// TIA Portal V19 export
FUNCTION "Decoiler1_CALL" : Void   // FC129, LAD
TITLE = DECOILER 1 CALL
// stored: SetENOAutomatically false
   VAR_TEMP
      Feed_PB_InLine : "Ax_PB";
      Feed_PB_OutLine : "Ax_PB";
      Jaws_PB_InLine : "ValveMachine_PB";
      Jaws_PB_OutLine : "ValveMachine_PB";
      Coupling_PB_InLine : "ValveMachine_PB";
      Coupling_PB_OutLine : "ValveMachine_PB";
      SnubberLift_PB_InLine : "ValveMachine_PB";
      SnubberLift_PB_OutLine : "ValveMachine_PB";
      SnubberRoll_PB_InLine : "ValveMachine_PB";
      SnubberRoll_PB_OutLine : "ValveMachine_PB";
   END_VAR
BEGIN

REGION Network 1: Data In - PB Feed
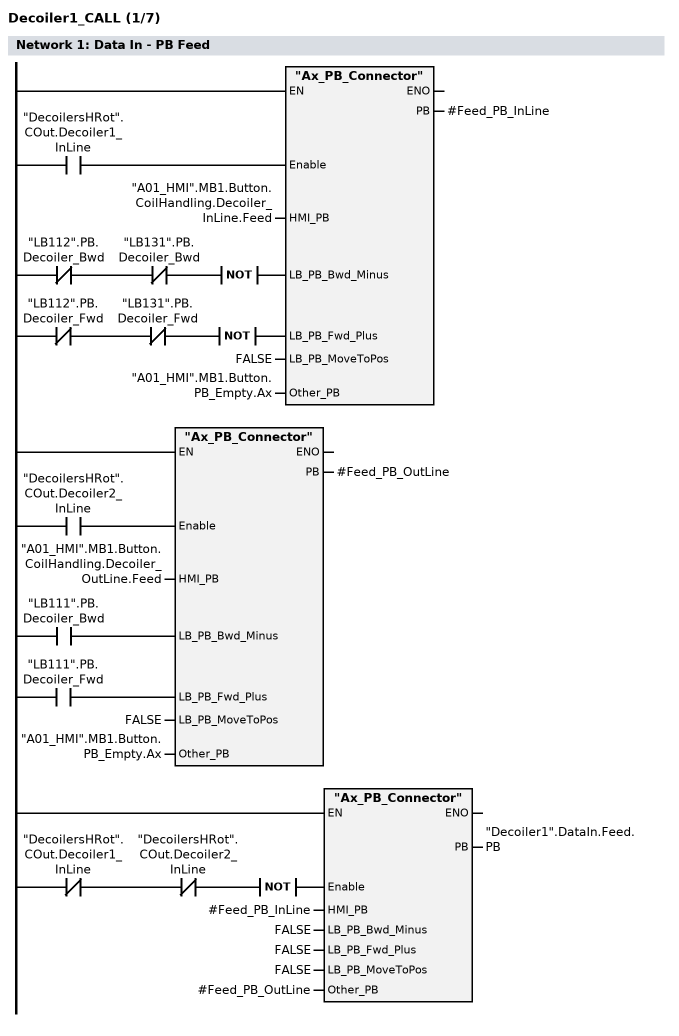
   RUNG wire#powerrail
      "Ax_PB_Connector"(Enable := wire#w1, LB_PB_Bwd_Minus := wire#w2, LB_PB_Fwd_Plus := wire#w3, HMI_PB := "A01_HMI".MB1.Button.CoilHandling.Decoiler_InLine.Feed, LB_PB_MoveToPos := FALSE, Other_PB := "A01_HMI".MB1.Button.PB_Empty.Ax, PB => #Feed_PB_InLine)
   END_RUNG
   RUNG wire#powerrail
      Contact( "DecoilersHRot".COut.Decoiler1_InLine )
   END_RUNG wire#w1
   RUNG wire#powerrail
      I_Contact( "LB112".PB.Decoiler_Bwd )
      I_Contact( "LB131".PB.Decoiler_Bwd )
      Not()
   END_RUNG wire#w2
   RUNG wire#powerrail
      I_Contact( "LB112".PB.Decoiler_Fwd )
      I_Contact( "LB131".PB.Decoiler_Fwd )
      Not()
   END_RUNG wire#w3
   RUNG wire#powerrail
      "Ax_PB_Connector"(Enable := wire#w4, LB_PB_Bwd_Minus := wire#w5, LB_PB_Fwd_Plus := wire#w6, HMI_PB := "A01_HMI".MB1.Button.CoilHandling.Decoiler_OutLine.Feed, LB_PB_MoveToPos := FALSE, Other_PB := "A01_HMI".MB1.Button.PB_Empty.Ax, PB => #Feed_PB_OutLine)
   END_RUNG
   RUNG wire#powerrail
      Contact( "DecoilersHRot".COut.Decoiler2_InLine )
   END_RUNG wire#w4
   RUNG wire#powerrail
      Contact( "LB111".PB.Decoiler_Bwd )
   END_RUNG wire#w5
   RUNG wire#powerrail
      Contact( "LB111".PB.Decoiler_Fwd )
   END_RUNG wire#w6
   RUNG wire#powerrail
      "Ax_PB_Connector"(Enable := wire#w7, HMI_PB := #Feed_PB_InLine, LB_PB_Bwd_Minus := FALSE, LB_PB_Fwd_Plus := FALSE, LB_PB_MoveToPos := FALSE, Other_PB := #Feed_PB_OutLine, PB => "Decoiler1".DataIn.Feed.PB)
   END_RUNG
   RUNG wire#powerrail
      I_Contact( "DecoilersHRot".COut.Decoiler1_InLine )
      I_Contact( "DecoilersHRot".COut.Decoiler2_InLine )
      Not()
   END_RUNG wire#w7
   // the same network as SCL:
   "Ax_PB_Connector"(Enable := "DecoilersHRot".COut.Decoiler1_InLine,
                     HMI_PB := "A01_HMI".MB1.Button.CoilHandling.Decoiler_InLine.Feed,
                     LB_PB_Bwd_Minus := NOT (NOT "LB112".PB.Decoiler_Bwd AND NOT "LB131".PB.Decoiler_Bwd),
                     LB_PB_Fwd_Plus := NOT (NOT "LB112".PB.Decoiler_Fwd AND NOT "LB131".PB.Decoiler_Fwd),
                     LB_PB_MoveToPos := FALSE,
                     Other_PB := "A01_HMI".MB1.Button.PB_Empty.Ax,
                     PB => #Feed_PB_InLine);
   "Ax_PB_Connector"(Enable := "DecoilersHRot".COut.Decoiler2_InLine,
                     HMI_PB := "A01_HMI".MB1.Button.CoilHandling.Decoiler_OutLine.Feed,
                     LB_PB_Bwd_Minus := "LB111".PB.Decoiler_Bwd,
                     LB_PB_Fwd_Plus := "LB111".PB.Decoiler_Fwd,
                     LB_PB_MoveToPos := FALSE,
                     Other_PB := "A01_HMI".MB1.Button.PB_Empty.Ax,
                     PB => #Feed_PB_OutLine);
   "Ax_PB_Connector"(Enable := NOT (NOT "DecoilersHRot".COut.Decoiler1_InLine AND NOT "DecoilersHRot".COut.Decoiler2_InLine),
                     HMI_PB := #Feed_PB_InLine,
                     LB_PB_Bwd_Minus := FALSE,
                     LB_PB_Fwd_Plus := FALSE,
                     LB_PB_MoveToPos := FALSE,
                     Other_PB := #Feed_PB_OutLine,
                     PB => "Decoiler1".DataIn.Feed.PB);
END_REGION

REGION Network 2: Data In - PB Jaws
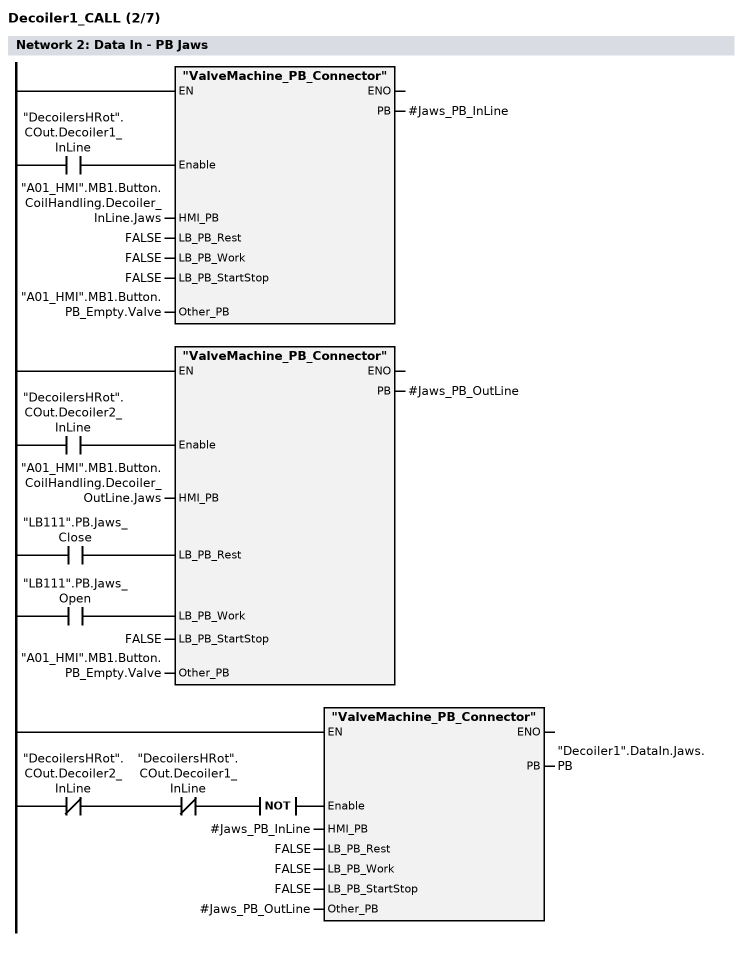
   RUNG wire#powerrail
      "ValveMachine_PB_Connector"(Enable := wire#w1, HMI_PB := "A01_HMI".MB1.Button.CoilHandling.Decoiler_InLine.Jaws, LB_PB_Rest := FALSE, LB_PB_Work := FALSE, LB_PB_StartStop := FALSE, Other_PB := "A01_HMI".MB1.Button.PB_Empty.Valve, PB => #Jaws_PB_InLine)
   END_RUNG
   RUNG wire#powerrail
      Contact( "DecoilersHRot".COut.Decoiler1_InLine )
   END_RUNG wire#w1
   RUNG wire#powerrail
      "ValveMachine_PB_Connector"(Enable := wire#w2, LB_PB_Rest := wire#w3, LB_PB_Work := wire#w4, HMI_PB := "A01_HMI".MB1.Button.CoilHandling.Decoiler_OutLine.Jaws, LB_PB_StartStop := FALSE, Other_PB := "A01_HMI".MB1.Button.PB_Empty.Valve, PB => #Jaws_PB_OutLine)
   END_RUNG
   RUNG wire#powerrail
      Contact( "DecoilersHRot".COut.Decoiler2_InLine )
   END_RUNG wire#w2
   RUNG wire#powerrail
      Contact( "LB111".PB.Jaws_Close )
   END_RUNG wire#w3
   RUNG wire#powerrail
      Contact( "LB111".PB.Jaws_Open )
   END_RUNG wire#w4
   RUNG wire#powerrail
      "ValveMachine_PB_Connector"(Enable := wire#w5, HMI_PB := #Jaws_PB_InLine, LB_PB_Rest := FALSE, LB_PB_Work := FALSE, LB_PB_StartStop := FALSE, Other_PB := #Jaws_PB_OutLine, PB => "Decoiler1".DataIn.Jaws.PB)
   END_RUNG
   RUNG wire#powerrail
      I_Contact( "DecoilersHRot".COut.Decoiler2_InLine )
      I_Contact( "DecoilersHRot".COut.Decoiler1_InLine )
      Not()
   END_RUNG wire#w5
   // the same network as SCL:
   "ValveMachine_PB_Connector"(Enable := "DecoilersHRot".COut.Decoiler1_InLine,
                           HMI_PB := "A01_HMI".MB1.Button.CoilHandling.Decoiler_InLine.Jaws,
                           LB_PB_Rest := FALSE,
                           LB_PB_Work := FALSE,
                           LB_PB_StartStop := FALSE,
                           Other_PB := "A01_HMI".MB1.Button.PB_Empty.Valve,
                           PB => #Jaws_PB_InLine);
   "ValveMachine_PB_Connector"(Enable := "DecoilersHRot".COut.Decoiler2_InLine,
                           HMI_PB := "A01_HMI".MB1.Button.CoilHandling.Decoiler_OutLine.Jaws,
                           LB_PB_Rest := "LB111".PB.Jaws_Close,
                           LB_PB_Work := "LB111".PB.Jaws_Open,
                           LB_PB_StartStop := FALSE,
                           Other_PB := "A01_HMI".MB1.Button.PB_Empty.Valve,
                           PB => #Jaws_PB_OutLine);
   "ValveMachine_PB_Connector"(Enable := NOT (NOT "DecoilersHRot".COut.Decoiler2_InLine AND NOT "DecoilersHRot".COut.Decoiler1_InLine),
                           HMI_PB := #Jaws_PB_InLine,
                           LB_PB_Rest := FALSE,
                           LB_PB_Work := FALSE,
                           LB_PB_StartStop := FALSE,
                           Other_PB := #Jaws_PB_OutLine,
                           PB => "Decoiler1".DataIn.Jaws.PB);
END_REGION

REGION Network 3: Data In - PB Couplung
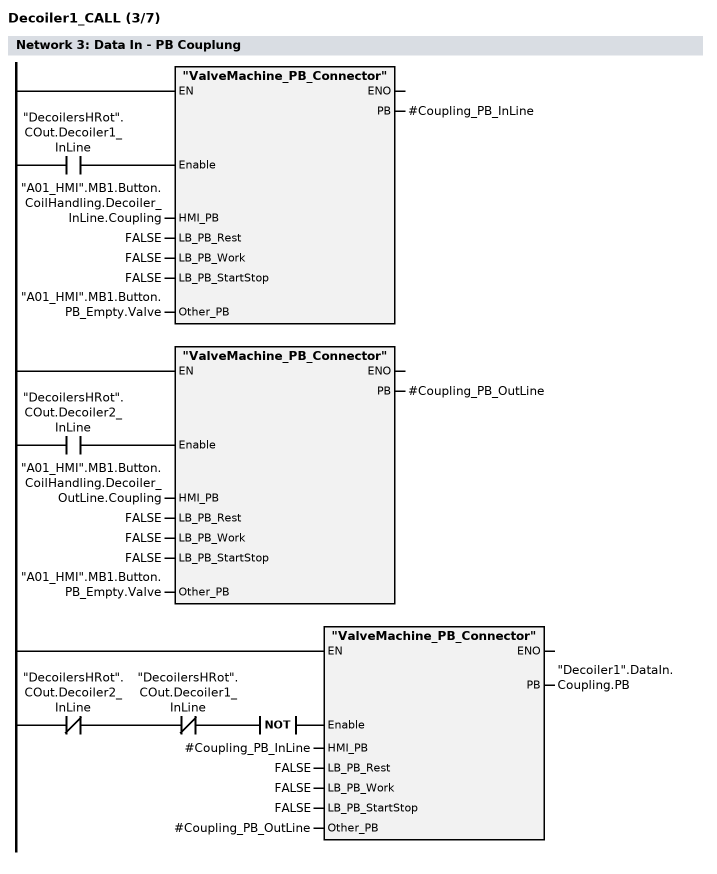
   RUNG wire#powerrail
      "ValveMachine_PB_Connector"(Enable := wire#w1, HMI_PB := "A01_HMI".MB1.Button.CoilHandling.Decoiler_InLine.Coupling, LB_PB_Rest := FALSE, LB_PB_Work := FALSE, LB_PB_StartStop := FALSE, Other_PB := "A01_HMI".MB1.Button.PB_Empty.Valve, PB => #Coupling_PB_InLine)
   END_RUNG
   RUNG wire#powerrail
      Contact( "DecoilersHRot".COut.Decoiler1_InLine )
   END_RUNG wire#w1
   RUNG wire#powerrail
      "ValveMachine_PB_Connector"(Enable := wire#w2, HMI_PB := "A01_HMI".MB1.Button.CoilHandling.Decoiler_OutLine.Coupling, LB_PB_Rest := FALSE, LB_PB_Work := FALSE, LB_PB_StartStop := FALSE, Other_PB := "A01_HMI".MB1.Button.PB_Empty.Valve, PB => #Coupling_PB_OutLine)
   END_RUNG
   RUNG wire#powerrail
      Contact( "DecoilersHRot".COut.Decoiler2_InLine )
   END_RUNG wire#w2
   RUNG wire#powerrail
      "ValveMachine_PB_Connector"(Enable := wire#w3, HMI_PB := #Coupling_PB_InLine, LB_PB_Rest := FALSE, LB_PB_Work := FALSE, LB_PB_StartStop := FALSE, Other_PB := #Coupling_PB_OutLine, PB => "Decoiler1".DataIn.Coupling.PB)
   END_RUNG
   RUNG wire#powerrail
      I_Contact( "DecoilersHRot".COut.Decoiler2_InLine )
      I_Contact( "DecoilersHRot".COut.Decoiler1_InLine )
      Not()
   END_RUNG wire#w3
   // the same network as SCL:
   "ValveMachine_PB_Connector"(Enable := "DecoilersHRot".COut.Decoiler1_InLine,
                           HMI_PB := "A01_HMI".MB1.Button.CoilHandling.Decoiler_InLine.Coupling,
                           LB_PB_Rest := FALSE,
                           LB_PB_Work := FALSE,
                           LB_PB_StartStop := FALSE,
                           Other_PB := "A01_HMI".MB1.Button.PB_Empty.Valve,
                           PB => #Coupling_PB_InLine);
   "ValveMachine_PB_Connector"(Enable := "DecoilersHRot".COut.Decoiler2_InLine,
                           HMI_PB := "A01_HMI".MB1.Button.CoilHandling.Decoiler_OutLine.Coupling,
                           LB_PB_Rest := FALSE,
                           LB_PB_Work := FALSE,
                           LB_PB_StartStop := FALSE,
                           Other_PB := "A01_HMI".MB1.Button.PB_Empty.Valve,
                           PB => #Coupling_PB_OutLine);
   "ValveMachine_PB_Connector"(Enable := NOT (NOT "DecoilersHRot".COut.Decoiler2_InLine AND NOT "DecoilersHRot".COut.Decoiler1_InLine),
                           HMI_PB := #Coupling_PB_InLine,
                           LB_PB_Rest := FALSE,
                           LB_PB_Work := FALSE,
                           LB_PB_StartStop := FALSE,
                           Other_PB := #Coupling_PB_OutLine,
                           PB => "Decoiler1".DataIn.Coupling.PB);
END_REGION

REGION Network 4: Data In - PB Snubber Lift
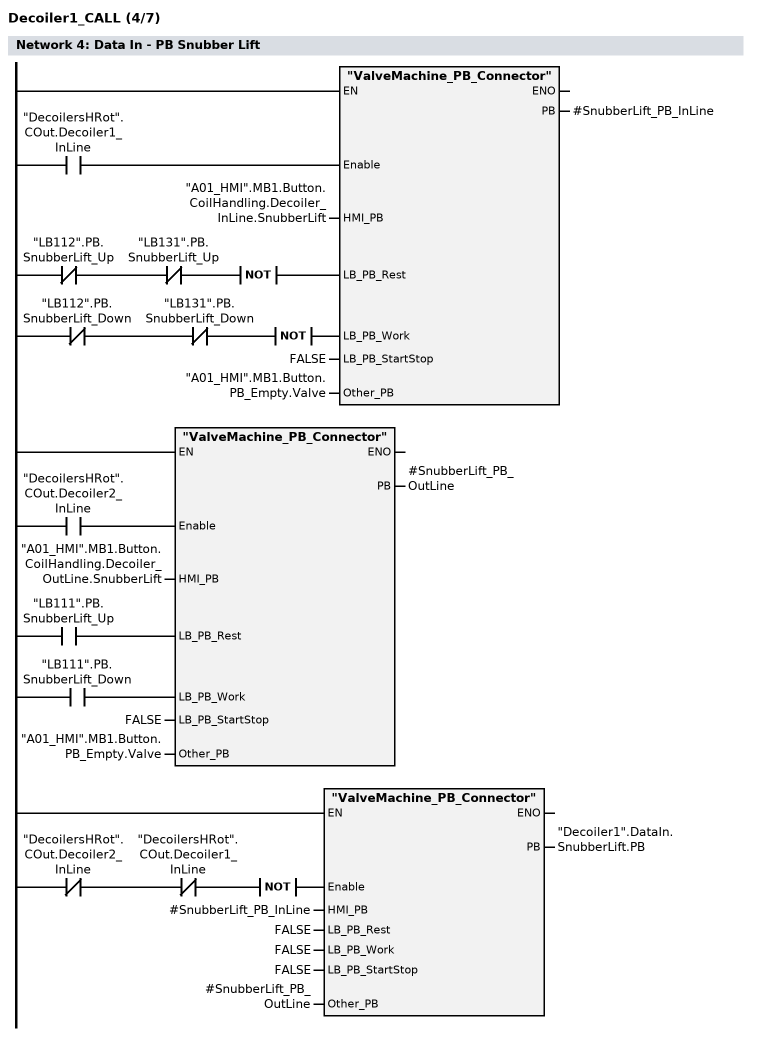
   RUNG wire#powerrail
      "ValveMachine_PB_Connector"(Enable := wire#w1, LB_PB_Rest := wire#w2, LB_PB_Work := wire#w3, HMI_PB := "A01_HMI".MB1.Button.CoilHandling.Decoiler_InLine.SnubberLift, LB_PB_StartStop := FALSE, Other_PB := "A01_HMI".MB1.Button.PB_Empty.Valve, PB => #SnubberLift_PB_InLine)
   END_RUNG
   RUNG wire#powerrail
      Contact( "DecoilersHRot".COut.Decoiler1_InLine )
   END_RUNG wire#w1
   RUNG wire#powerrail
      I_Contact( "LB112".PB.SnubberLift_Up )
      I_Contact( "LB131".PB.SnubberLift_Up )
      Not()
   END_RUNG wire#w2
   RUNG wire#powerrail
      I_Contact( "LB112".PB.SnubberLift_Down )
      I_Contact( "LB131".PB.SnubberLift_Down )
      Not()
   END_RUNG wire#w3
   RUNG wire#powerrail
      "ValveMachine_PB_Connector"(Enable := wire#w4, LB_PB_Rest := wire#w5, LB_PB_Work := wire#w6, HMI_PB := "A01_HMI".MB1.Button.CoilHandling.Decoiler_OutLine.SnubberLift, LB_PB_StartStop := FALSE, Other_PB := "A01_HMI".MB1.Button.PB_Empty.Valve, PB => #SnubberLift_PB_OutLine)
   END_RUNG
   RUNG wire#powerrail
      Contact( "DecoilersHRot".COut.Decoiler2_InLine )
   END_RUNG wire#w4
   RUNG wire#powerrail
      Contact( "LB111".PB.SnubberLift_Up )
   END_RUNG wire#w5
   RUNG wire#powerrail
      Contact( "LB111".PB.SnubberLift_Down )
   END_RUNG wire#w6
   RUNG wire#powerrail
      "ValveMachine_PB_Connector"(Enable := wire#w7, HMI_PB := #SnubberLift_PB_InLine, LB_PB_Rest := FALSE, LB_PB_Work := FALSE, LB_PB_StartStop := FALSE, Other_PB := #SnubberLift_PB_OutLine, PB => "Decoiler1".DataIn.SnubberLift.PB)
   END_RUNG
   RUNG wire#powerrail
      I_Contact( "DecoilersHRot".COut.Decoiler2_InLine )
      I_Contact( "DecoilersHRot".COut.Decoiler1_InLine )
      Not()
   END_RUNG wire#w7
   // the same network as SCL:
   "ValveMachine_PB_Connector"(Enable := "DecoilersHRot".COut.Decoiler1_InLine,
                           HMI_PB := "A01_HMI".MB1.Button.CoilHandling.Decoiler_InLine.SnubberLift,
                           LB_PB_Rest := NOT (NOT "LB112".PB.SnubberLift_Up AND NOT "LB131".PB.SnubberLift_Up),
                           LB_PB_Work := NOT (NOT "LB112".PB.SnubberLift_Down AND NOT "LB131".PB.SnubberLift_Down),
                           LB_PB_StartStop := FALSE,
                           Other_PB := "A01_HMI".MB1.Button.PB_Empty.Valve,
                           PB => #SnubberLift_PB_InLine);
   "ValveMachine_PB_Connector"(Enable := "DecoilersHRot".COut.Decoiler2_InLine,
                           HMI_PB := "A01_HMI".MB1.Button.CoilHandling.Decoiler_OutLine.SnubberLift,
                           LB_PB_Rest := "LB111".PB.SnubberLift_Up,
                           LB_PB_Work := "LB111".PB.SnubberLift_Down,
                           LB_PB_StartStop := FALSE,
                           Other_PB := "A01_HMI".MB1.Button.PB_Empty.Valve,
                           PB => #SnubberLift_PB_OutLine);
   "ValveMachine_PB_Connector"(Enable := NOT (NOT "DecoilersHRot".COut.Decoiler2_InLine AND NOT "DecoilersHRot".COut.Decoiler1_InLine),
                           HMI_PB := #SnubberLift_PB_InLine,
                           LB_PB_Rest := FALSE,
                           LB_PB_Work := FALSE,
                           LB_PB_StartStop := FALSE,
                           Other_PB := #SnubberLift_PB_OutLine,
                           PB => "Decoiler1".DataIn.SnubberLift.PB);
END_REGION

REGION Network 5: Data In - Snubber Roll
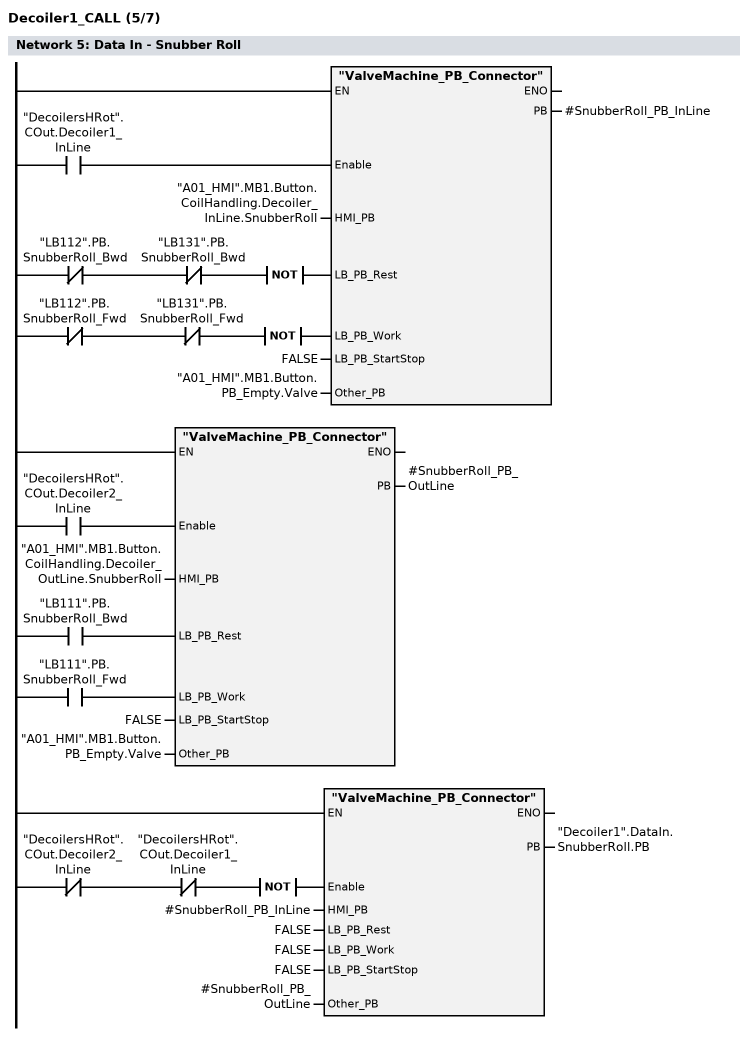
   RUNG wire#powerrail
      "ValveMachine_PB_Connector"(Enable := wire#w1, LB_PB_Rest := wire#w2, LB_PB_Work := wire#w3, HMI_PB := "A01_HMI".MB1.Button.CoilHandling.Decoiler_InLine.SnubberRoll, LB_PB_StartStop := FALSE, Other_PB := "A01_HMI".MB1.Button.PB_Empty.Valve, PB => #SnubberRoll_PB_InLine)
   END_RUNG
   RUNG wire#powerrail
      Contact( "DecoilersHRot".COut.Decoiler1_InLine )
   END_RUNG wire#w1
   RUNG wire#powerrail
      I_Contact( "LB112".PB.SnubberRoll_Bwd )
      I_Contact( "LB131".PB.SnubberRoll_Bwd )
      Not()
   END_RUNG wire#w2
   RUNG wire#powerrail
      I_Contact( "LB112".PB.SnubberRoll_Fwd )
      I_Contact( "LB131".PB.SnubberRoll_Fwd )
      Not()
   END_RUNG wire#w3
   RUNG wire#powerrail
      "ValveMachine_PB_Connector"(Enable := wire#w4, LB_PB_Rest := wire#w5, LB_PB_Work := wire#w6, HMI_PB := "A01_HMI".MB1.Button.CoilHandling.Decoiler_OutLine.SnubberRoll, LB_PB_StartStop := FALSE, Other_PB := "A01_HMI".MB1.Button.PB_Empty.Valve, PB => #SnubberRoll_PB_OutLine)
   END_RUNG
   RUNG wire#powerrail
      Contact( "DecoilersHRot".COut.Decoiler2_InLine )
   END_RUNG wire#w4
   RUNG wire#powerrail
      Contact( "LB111".PB.SnubberRoll_Bwd )
   END_RUNG wire#w5
   RUNG wire#powerrail
      Contact( "LB111".PB.SnubberRoll_Fwd )
   END_RUNG wire#w6
   RUNG wire#powerrail
      "ValveMachine_PB_Connector"(Enable := wire#w7, HMI_PB := #SnubberRoll_PB_InLine, LB_PB_Rest := FALSE, LB_PB_Work := FALSE, LB_PB_StartStop := FALSE, Other_PB := #SnubberRoll_PB_OutLine, PB => "Decoiler1".DataIn.SnubberRoll.PB)
   END_RUNG
   RUNG wire#powerrail
      I_Contact( "DecoilersHRot".COut.Decoiler2_InLine )
      I_Contact( "DecoilersHRot".COut.Decoiler1_InLine )
      Not()
   END_RUNG wire#w7
   // the same network as SCL:
   "ValveMachine_PB_Connector"(Enable := "DecoilersHRot".COut.Decoiler1_InLine,
                           HMI_PB := "A01_HMI".MB1.Button.CoilHandling.Decoiler_InLine.SnubberRoll,
                           LB_PB_Rest := NOT (NOT "LB112".PB.SnubberRoll_Bwd AND NOT "LB131".PB.SnubberRoll_Bwd),
                           LB_PB_Work := NOT (NOT "LB112".PB.SnubberRoll_Fwd AND NOT "LB131".PB.SnubberRoll_Fwd),
                           LB_PB_StartStop := FALSE,
                           Other_PB := "A01_HMI".MB1.Button.PB_Empty.Valve,
                           PB => #SnubberRoll_PB_InLine);
   "ValveMachine_PB_Connector"(Enable := "DecoilersHRot".COut.Decoiler2_InLine,
                           HMI_PB := "A01_HMI".MB1.Button.CoilHandling.Decoiler_OutLine.SnubberRoll,
                           LB_PB_Rest := "LB111".PB.SnubberRoll_Bwd,
                           LB_PB_Work := "LB111".PB.SnubberRoll_Fwd,
                           LB_PB_StartStop := FALSE,
                           Other_PB := "A01_HMI".MB1.Button.PB_Empty.Valve,
                           PB => #SnubberRoll_PB_OutLine);
   "ValveMachine_PB_Connector"(Enable := NOT (NOT "DecoilersHRot".COut.Decoiler2_InLine AND NOT "DecoilersHRot".COut.Decoiler1_InLine),
                           HMI_PB := #SnubberRoll_PB_InLine,
                           LB_PB_Rest := FALSE,
                           LB_PB_Work := FALSE,
                           LB_PB_StartStop := FALSE,
                           Other_PB := #SnubberRoll_PB_OutLine,
                           PB => "Decoiler1".DataIn.SnubberRoll.PB);
END_REGION

REGION Network 6: Data In - Pneumatic Brake
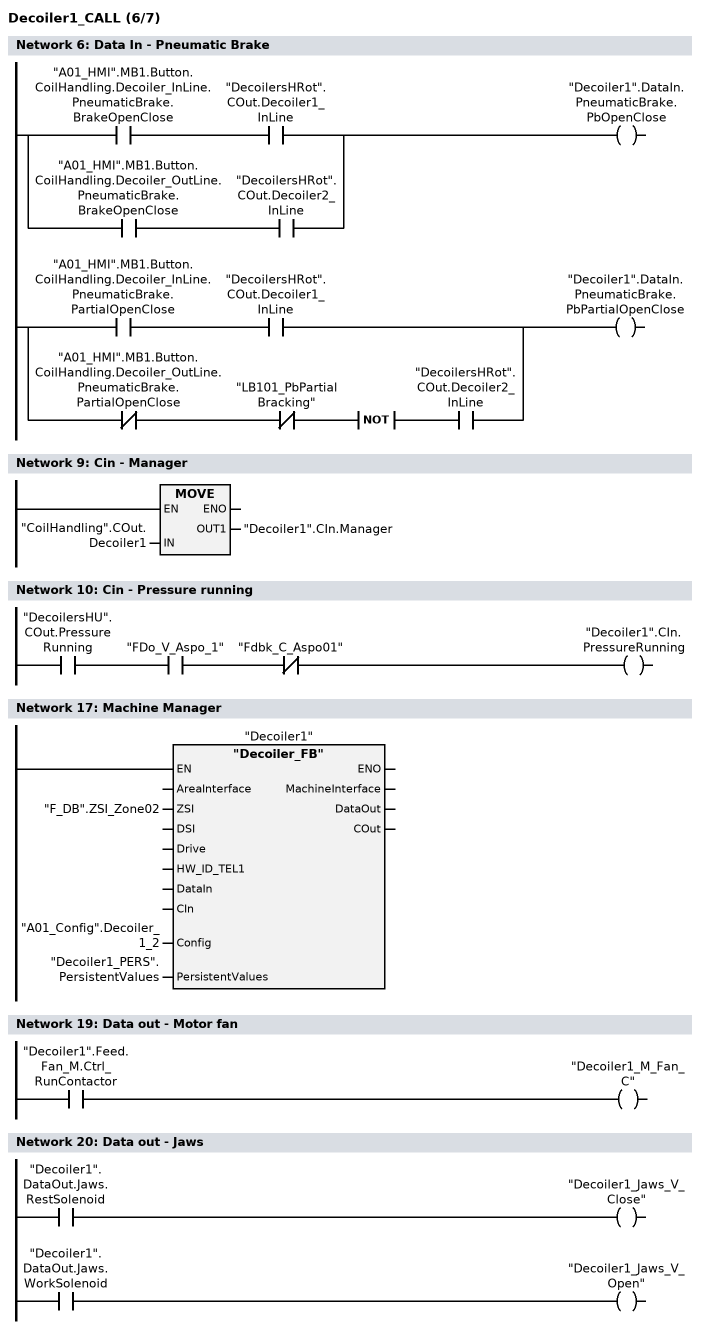
   RUNG wire#powerrail
      Contact( "A01_HMI".MB1.Button.CoilHandling.Decoiler_InLine.PneumaticBrake.BrakeOpenClose )
      Contact( "DecoilersHRot".COut.Decoiler1_InLine )
      wire#w1
      Coil( "Decoiler1".DataIn.PneumaticBrake.PbOpenClose )
   END_RUNG
   RUNG wire#powerrail
      Contact( "A01_HMI".MB1.Button.CoilHandling.Decoiler_OutLine.PneumaticBrake.BrakeOpenClose )
      Contact( "DecoilersHRot".COut.Decoiler2_InLine )
   END_RUNG wire#w1
   RUNG wire#powerrail
      Contact( "A01_HMI".MB1.Button.CoilHandling.Decoiler_InLine.PneumaticBrake.PartialOpenClose )
      Contact( "DecoilersHRot".COut.Decoiler1_InLine )
      wire#w2
      Coil( "Decoiler1".DataIn.PneumaticBrake.PbPartialOpenClose )
   END_RUNG
   RUNG wire#powerrail
      I_Contact( "A01_HMI".MB1.Button.CoilHandling.Decoiler_OutLine.PneumaticBrake.PartialOpenClose )
      I_Contact( "LB101_PbPartialBracking" )
      Not()
      Contact( "DecoilersHRot".COut.Decoiler2_InLine )
   END_RUNG wire#w2
   // the same network as SCL:
   "Decoiler1".DataIn.PneumaticBrake.PbOpenClose := ("A01_HMI".MB1.Button.CoilHandling.Decoiler_InLine.PneumaticBrake.BrakeOpenClose AND "DecoilersHRot".COut.Decoiler1_InLine) OR ("A01_HMI".MB1.Button.CoilHandling.Decoiler_OutLine.PneumaticBrake.BrakeOpenClose AND "DecoilersHRot".COut.Decoiler2_InLine);
   "Decoiler1".DataIn.PneumaticBrake.PbPartialOpenClose := ("A01_HMI".MB1.Button.CoilHandling.Decoiler_InLine.PneumaticBrake.PartialOpenClose AND "DecoilersHRot".COut.Decoiler1_InLine) OR (NOT (NOT "A01_HMI".MB1.Button.CoilHandling.Decoiler_OutLine.PneumaticBrake.PartialOpenClose AND NOT "LB101_PbPartialBracking") AND "DecoilersHRot".COut.Decoiler2_InLine);
END_REGION

REGION Network 7 (SCL): Data In - Sensors
   //Loop
   "Decoiler1".DataIn.DiameterSensor := "DecoilerX_AI_Coil_Diameter";
   "Decoiler1".DataIn.Loop.Connector := TRUE;



   "Decoiler1".DataIn.Loop.S_MinHigh := FALSE;
   "Decoiler1".DataIn.Loop.S_MaxLow := FALSE; 
   "Decoiler1".DataIn.Loop.S_SpeedAsjust := FALSE;


   IF  "A01_DEBUG".CoilHandling_Simulation.DecoilerInLine_Sensors.Enable
   THEN

       "Decoiler1".DataIn.Loop.S_MinHigh := "A01_DEBUG".CoilHandling_Simulation.DecoilerInLine_Sensors.Phc_Min;
       "Decoiler1".DataIn.Loop.S_MaxLow := "A01_DEBUG".CoilHandling_Simulation.DecoilerInLine_Sensors.Phc_Max;
     "Decoiler1".DataIn.Loop.S_SpeedAsjust := "A01_DEBUG".CoilHandling_Simulation.DecoilerInLine_Sensors.Phc_SpeedAdjust;


   END_IF;




   //Feed 
   "Decoiler1".DataIn.Feed.Fan_M_Feedback := "Decoiler1_M_Fan_Fdbk";



   //COupling
   "Decoiler1".DataIn.Coupling.Rest_Ls[1] := "Decoier1_Coupling_Ls_Rest";
   "Decoiler1".DataIn.Coupling.Work_Ls[1] := "Decoier1_Coupling_Ls_Work";

   //Snubber Lift
   "Decoiler1".DataIn.SnubberLift.Rest_Ls[1] := "Decoiler1_Snubber_Lift_Ls_UP";
END_REGION

REGION Network 8: >
END_REGION

REGION Network 9: Cin - Manager
   RUNG wire#powerrail
      Move(in := "CoilHandling".COut.Decoiler1, out1 => "Decoiler1".CIn.Manager)
   END_RUNG
   // the same network as SCL:
   "Decoiler1".CIn.Manager := "CoilHandling".COut.Decoiler1;
END_REGION

REGION Network 10: Cin - Pressure running
   RUNG wire#powerrail
      Contact( "DecoilersHU".COut.PressureRunning )
      Contact( "FDo_V_Aspo_1" )
      I_Contact( "Fdbk_C_Aspo01" )
      Coil( "Decoiler1".CIn.PressureRunning )
   END_RUNG
   // the same network as SCL:
   "Decoiler1".CIn.PressureRunning := "DecoilersHU".COut.PressureRunning AND "FDo_V_Aspo_1" AND NOT "Fdbk_C_Aspo01";
END_REGION

REGION Network 11: >
END_REGION

REGION Network 12 (SCL): Area interface

   "Decoiler1".AreaInterface := "Area01".AreaInterface;

   // Case IN-LINE
   IF "DecoilersHRot".COut.Decoiler1_InLine THEN

       "Decoiler1".AreaInterface := "Area01".AreaInterface;

   // Case OUT-LINE
   ELSIF "DecoilersHRot".COut.Decoiler2_InLine THEN


       "Decoiler1".AreaInterface.Man := NOT "Area01".AreaInterface.EStop;
       "Decoiler1".AreaInterface.Aut := FALSE;
       "Decoiler1".AreaInterface.Cycle := FALSE;
       "Decoiler1".AreaInterface.StopInPhase := FALSE;
       "Decoiler1".AreaInterface.StopProgrammed := FALSE;
       "Decoiler1".AreaInterface.CheckAutReady := FALSE;

   // Case UNKNOW
   // 
   ELSE

       "Decoiler1".AreaInterface.EStop := TRUE;
       "Decoiler1".AreaInterface.Man := FALSE;
       "Decoiler1".AreaInterface.Aut := FALSE;
       "Decoiler1".AreaInterface.Cycle := FALSE;

   END_IF;
END_REGION

REGION Network 13 (SCL): DSI
   "Decoiler1".DSI.Feed := "F_DB".DSI_S120_Decoiler1;

   "Decoiler1".DSI.Jaws :=
   "Decoiler1".DSI.Coupling :=
   "Decoiler1".DSI.SnubberLift :=
   "Decoiler1".DSI.SnubberRoll := "F_DB".DSI_V_Decoiler1;
END_REGION

REGION Network 14 (SCL): Drive
   "Decoiler1".Drive.Infeed_ON := "Areas_ITF".AG.Infeed_Running;
   "Decoiler1".Drive.AccessPoint := "HW_Const_Values".CU1_PN_740A1_1_ModuleAccessPoint;
   "Decoiler1".Drive.AxisID := "CU1_ID_3_740A1_1_740M1";
   "Decoiler1".Drive.TokenChain := "TOKENCHAIN_CU1";
END_REGION

REGION Network 15 (SCL): HW ID
   "Decoiler1".HW_ID_TEL1 := "HW_Const_Values".CU1_PN_740A1_1_Standard_telegram_1;
END_REGION

REGION Network 16: >
END_REGION

REGION Network 17: Machine Manager
   RUNG wire#powerrail
      "Decoiler1"(AreaInterface :=, ZSI := "F_DB".ZSI_Zone02, DSI :=, Drive :=, HW_ID_TEL1 :=, DataIn :=, CIn :=, Config := "A01_Config".Decoiler_1_2, PersistentValues := "Decoiler1_PERS".PersistentValues, MachineInterface =>, DataOut =>, COut =>)
   END_RUNG
   // the same network as SCL:
   "Decoiler1"(ZSI := "F_DB".ZSI_Zone02,   // "Decoiler_FB"
               Config := "A01_Config".Decoiler_1_2,
               PersistentValues := "Decoiler1_PERS".PersistentValues);
END_REGION

REGION Network 18: >
END_REGION

REGION Network 19: Data out - Motor fan
   RUNG wire#powerrail
      Contact( "Decoiler1".Feed.Fan_M.Ctrl_RunContactor )
      Coil( "Decoiler1_M_Fan_C" )
   END_RUNG
   // the same network as SCL:
   "Decoiler1_M_Fan_C" := "Decoiler1".Feed.Fan_M.Ctrl_RunContactor;
END_REGION

REGION Network 20: Data out - Jaws
   RUNG wire#powerrail
      Contact( "Decoiler1".DataOut.Jaws.RestSolenoid )
      Coil( "Decoiler1_Jaws_V_Close" )
   END_RUNG
   RUNG wire#powerrail
      Contact( "Decoiler1".DataOut.Jaws.WorkSolenoid )
      Coil( "Decoiler1_Jaws_V_Open" )
   END_RUNG
   // the same network as SCL:
   "Decoiler1_Jaws_V_Close" := "Decoiler1".DataOut.Jaws.RestSolenoid;
   "Decoiler1_Jaws_V_Open" := "Decoiler1".DataOut.Jaws.WorkSolenoid;
END_REGION

REGION Network 21: Data out - Motor coupling
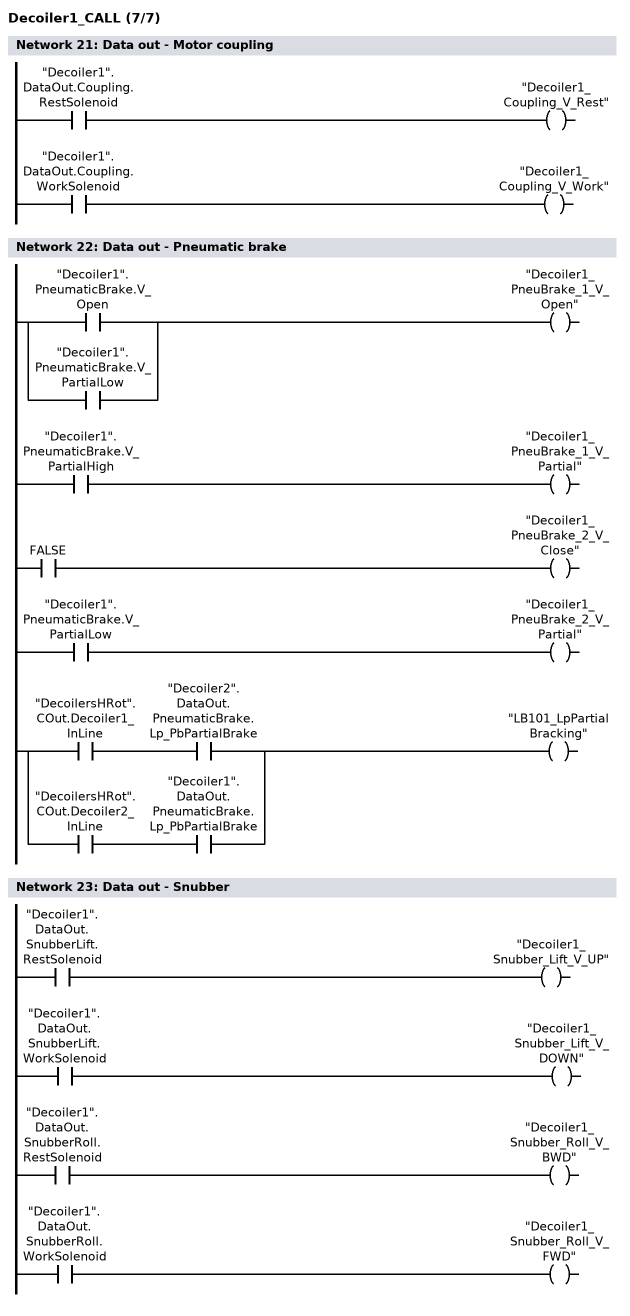
   RUNG wire#powerrail
      Contact( "Decoiler1".DataOut.Coupling.RestSolenoid )
      Coil( "Decoiler1_Coupling_V_Rest" )
   END_RUNG
   RUNG wire#powerrail
      Contact( "Decoiler1".DataOut.Coupling.WorkSolenoid )
      Coil( "Decoiler1_Coupling_V_Work" )
   END_RUNG
   // the same network as SCL:
   "Decoiler1_Coupling_V_Rest" := "Decoiler1".DataOut.Coupling.RestSolenoid;
   "Decoiler1_Coupling_V_Work" := "Decoiler1".DataOut.Coupling.WorkSolenoid;
END_REGION

REGION Network 22: Data out - Pneumatic brake
   RUNG wire#powerrail
      Contact( "Decoiler1".PneumaticBrake.V_Open )
      wire#w1
      Coil( "Decoiler1_PneuBrake_1_V_Open" )
   END_RUNG
   RUNG wire#powerrail
      Contact( "Decoiler1".PneumaticBrake.V_PartialLow )
   END_RUNG wire#w1
   RUNG wire#powerrail
      Contact( "Decoiler1".PneumaticBrake.V_PartialHigh )
      Coil( "Decoiler1_PneuBrake_1_V_Partial" )
   END_RUNG
   RUNG wire#powerrail
      Contact( FALSE )
      Coil( "Decoiler1_PneuBrake_2_V_Close" )
   END_RUNG
   RUNG wire#powerrail
      Contact( "Decoiler1".PneumaticBrake.V_PartialLow )
      Coil( "Decoiler1_PneuBrake_2_V_Partial" )
   END_RUNG
   RUNG wire#powerrail
      Contact( "DecoilersHRot".COut.Decoiler1_InLine )
      Contact( "Decoiler2".DataOut.PneumaticBrake.Lp_PbPartialBrake )
      wire#w2
      Coil( "LB101_LpPartialBracking" )
   END_RUNG
   RUNG wire#powerrail
      Contact( "DecoilersHRot".COut.Decoiler2_InLine )
      Contact( "Decoiler1".DataOut.PneumaticBrake.Lp_PbPartialBrake )
   END_RUNG wire#w2
   // the same network as SCL:
   "Decoiler1_PneuBrake_1_V_Open" := "Decoiler1".PneumaticBrake.V_Open OR "Decoiler1".PneumaticBrake.V_PartialLow;
   "Decoiler1_PneuBrake_1_V_Partial" := "Decoiler1".PneumaticBrake.V_PartialHigh;
   "Decoiler1_PneuBrake_2_V_Close" := FALSE;
   "Decoiler1_PneuBrake_2_V_Partial" := "Decoiler1".PneumaticBrake.V_PartialLow;
   "LB101_LpPartialBracking" := ("DecoilersHRot".COut.Decoiler1_InLine AND "Decoiler2".DataOut.PneumaticBrake.Lp_PbPartialBrake) OR ("DecoilersHRot".COut.Decoiler2_InLine AND "Decoiler1".DataOut.PneumaticBrake.Lp_PbPartialBrake);
END_REGION

REGION Network 23: Data out - Snubber
   RUNG wire#powerrail
      Contact( "Decoiler1".DataOut.SnubberLift.RestSolenoid )
      Coil( "Decoiler1_Snubber_Lift_V_UP" )
   END_RUNG
   RUNG wire#powerrail
      Contact( "Decoiler1".DataOut.SnubberLift.WorkSolenoid )
      Coil( "Decoiler1_Snubber_Lift_V_DOWN" )
   END_RUNG
   RUNG wire#powerrail
      Contact( "Decoiler1".DataOut.SnubberRoll.RestSolenoid )
      Coil( "Decoiler1_Snubber_Roll_V_BWD" )
   END_RUNG
   RUNG wire#powerrail
      Contact( "Decoiler1".DataOut.SnubberRoll.WorkSolenoid )
      Coil( "Decoiler1_Snubber_Roll_V_FWD" )
   END_RUNG
   // the same network as SCL:
   "Decoiler1_Snubber_Lift_V_UP" := "Decoiler1".DataOut.SnubberLift.RestSolenoid;
   "Decoiler1_Snubber_Lift_V_DOWN" := "Decoiler1".DataOut.SnubberLift.WorkSolenoid;
   "Decoiler1_Snubber_Roll_V_BWD" := "Decoiler1".DataOut.SnubberRoll.RestSolenoid;
   "Decoiler1_Snubber_Roll_V_FWD" := "Decoiler1".DataOut.SnubberRoll.WorkSolenoid;
END_REGION

REGION Network 24: >
END_REGION

REGION Network 25: >
END_REGION

REGION Network 26: >
END_REGION
END_FUNCTION
